FUNCTION_BLOCK Test_1
VAR_INPUT
END_VAR
VAR_OUTPUT
END_VAR
VAR
	heyo : REAL;
	random: BOOL;
	io				: ST_ProfinetDiagnostics;
	
END_VAR

random := not random;

PROPERTY P_IO : REFERENCE TO ST_ProfinetDiagnostics
GET
P_IO REF= io;
END_GET
END_PROPERTY

PROPERTY PUBLIC P_REAL : REFERENCE TO REAL
GET
P_REAL REF= heyo;
END_GET
END_PROPERTY

END_FUNCTION_BLOCK

(* stored: Version 1.1.0.1, ProductVersion 3.1.4024.12
   POU Test_1: Id {fa1ed945-89f6-4ed4-b3ce-2ab3f9743574}, SpecialFunc None
   Property P_IO: Id {e0dd2748-6ad2-4dde-8522-d0a99a3f5dfd}
   Get Get: Id {b2dfdf14-f359-4846-a826-c33a2ee06640}
   Property P_REAL: Id {c36ddca3-5e7e-4a68-b180-064903a74aea}
   Get Get: Id {f16b57d5-ff0f-42f4-983b-0bd3b57f2d8b} *)
